// TIA Portal V21 export
DATA_BLOCK "DB616"   // DB616
TITLE = DB616
{ S7_Optimized_Access := 'FALSE' }
// CIP Recipe
// stored: AutoNumber false
   VAR
      TotalStep : Int := 3;
      CycleSelection { S7_SetPoint := 'True'} : Array[0..3] of "CIP";
      MainPopup1Enable : Bool := 1;
      MainPopup2Enable : Bool := 1;
      FillingInputPara { S7_SetPoint := 'True'} : Array[0..3] of "FillingInputs";
      FillingOutputPara { S7_SetPoint := 'True'} : Array[0..3] of "FillingOutputs";
      MixingTimeInput : Array[0..3] of Int;
      RecirculationInput { S7_SetPoint := 'True'} : Array[0..3] of "RecirculationInputs";
      RecirculationOutput { S7_SetPoint := 'True'} : Array[0..3] of "RecirculationOutputs";
      DrainInputs { S7_SetPoint := 'True'} : Array[0..3] of "DrainInputs";
      DrainOutputs : Array[0..3] of "DrainOutputs";
      SystemDrainSetTimeInput : Array[0..3] of Int;
      SystemDrainOutPara { S7_SetPoint := 'True'} : Array[0..3] of "SystemDrainOutputs";
      AirPurgingInputPara { S7_SetPoint := 'True'} : Array[0..3] of "AirPurgingInputs";
      AirPurgingOutPara { S7_SetPoint := 'True'} : Array[0..3] of "AirPurgingOutputs";
      CycleNames : Array[0..3] of String[60];
      Spare : Bool;
   END_VAR
BEGIN
   CycleSelection[0..3].StepSelection.SuctionLineCleanNoYes := 0;
   CycleSelection[0..3].StepSelection.VacuumDryingNoYes := 0;
   CycleSelection[0].StepSelection.FillingNoYes := 0;
   CycleSelection[1..3].StepSelection.FillingNoYes := 1;
   CycleSelection[0..3].StepSelection.TemperatureDosingNoYes := 0;
   CycleSelection[0..3].StepSelection.TransferNoYes := 0;
   CycleSelection[0..1].StepSelection.MIxingNoYes := 0;
   CycleSelection[2..3].StepSelection.MIxingNoYes := 1;
   CycleSelection[0..1].StepSelection.RecirculationNoYes := 0;
   CycleSelection[2..3].StepSelection.RecirculationNoYes := 1;
   CycleSelection[0].StepSelection.DrainNoYes := 0;
   CycleSelection[1..3].StepSelection.DrainNoYes := 1;
   CycleSelection[0].StepSelection.SystemDrainNoYes := 0;
   CycleSelection[1..3].StepSelection.SystemDrainNoYes := 1;
   CycleSelection[0].StepSelection.AirPurgingNoYes := 0;
   CycleSelection[1..3].StepSelection.AirPurgingNoYes := 1;
   CycleSelection[1..3].StepSelection.ConductivityCheckWhileRinse := 0;
   CycleSelection[0..2].StepSelection.ConductivityCheckWhileDrain := 0;
   CycleSelection[3].StepSelection.ConductivityCheckWhileDrain := 1;
   CycleSelection[0..2].StepSelection.SetRepetition := 0;
   CycleSelection[0..3].StepSelection.TimeSaveModeNoYes := 0;
   CycleSelection[1].StepSelection.ConductivityCheckWhileTransfer := false;
   CycleSelection[2..3].StepSelection.ConductivityCheckWhileTransfer := 0;
   FillingInputPara[1].Selections.FillMethodSel := 3;
   FillingInputPara[2..3].Selections.FillMethodSel := 0;
   FillingInputPara[1..3].Selections.FillTimeBaseSel := 0;
   FillingInputPara[0].Selections.UtilitySel := 1;
   FillingInputPara[1..3].Selections.UtilitySel := 2;
   FillingInputPara[1..3].Selections.ConductivityWhileRinse := 0;
   FillingInputPara[0].Selections.RinseCondition := 1;
   FillingInputPara[1..3].Selections.RinseCondition := 0;
   FillingInputPara[1].Selections.BypassRinseCondition := 1;
   FillingInputPara[2..3].Selections.BypassRinseCondition := 0;
   FillingInputPara[1..3].Selections.BypassWeightWhileRinseCycle := 0;
   FillingInputPara[0..3].Selections.SeperateParaForRep := 1;
   FillingInputPara[1..2].ProductionSetting.LoopDelay1 := 0;
   FillingInputPara[1].ProductionSetting.ZDVDelay := 0;
   FillingInputPara[0].PreciseEngineering.Loops := 1;
   FillingInputPara[1].PreciseEngineering.Loops := 16;
   FillingInputPara[2..3].PreciseEngineering.Loops := 5;
   FillingInputPara[1..3].PreciseEngineering.VesselMaxWeight := 3000.0;
   MixingTimeInput[2..3] := 1;
   RecirculationInput[2..3].Selections.PressureModeSel := 0;
   RecirculationInput[2..3].Selections.PumpSel := 0;
   RecirculationInput[2].Parameters.RecirculationInputToRunTime := 0;
   RecirculationInput[1].PreciseEngineering.Loops := 0;
   RecirculationInput[2..3].PreciseEngineering.Loops := 5;
   DrainInputs[0..3].Selections.DrainMethodSel := 0;
   DrainInputs[1..3].Selections.PressureModeSel := 1;
   DrainInputs[1].Selections.DrainPumpSel := 0;
   DrainInputs[2..3].Selections.DrainPumpSel := 1;
   DrainInputs[0..1].Selections.InputToRunPump := 0;
   DrainInputs[2..3].Selections.InputToRunPump := 1;
   DrainInputs[1..2].Selections.ConductivityWhileDrain := 0;
   DrainInputs[3].Selections.ConductivityWhileDrain := 1;
   DrainInputs[1..2].Selections.ConductivityWhileDrainPTL := 0;
   DrainInputs[1..2].Selections.CipSkidWeightSel := 0;
   DrainInputs[1..2].Selections.MultiConductivityCheck := 0;
   DrainInputs[0..1].PreciseEngineering.Loops := 1;
   DrainInputs[2..3].PreciseEngineering.Loops := 10;
   AirPurgingInputPara[1..3].Selections.ApMethod := 0;
   AirPurgingInputPara[1..3].Selections.PressureMode := 1;
   AirPurgingInputPara[1..3].Selections.VentBeforeOver := 1;
   AirPurgingInputPara[1..3].Selections.AirPurgingSel := 0;
   AirPurgingInputPara[1..3].PreciseEngineering.Loops := 17;
   CycleNames[1] := 'PRE RINSE CYCLE';
   CycleNames[2] := 'FILLING CYCLE';
   CycleNames[3] := 'FINAL RINSE CYCLE';
END_DATA_BLOCK
